// TwinCAT 3 PLC project PLC2
// ProgramVersion: 3.1.4024.0
// libraries:
//   Tc2_Standard, * (Beckhoff Automation GmbH)
//   Tc2_System, * (Beckhoff Automation GmbH)
//   Tc3_Module, * (Beckhoff Automation GmbH)
// project tree:
//   GVLs/ GVL_Alarm.TcGVL
//   / PlcTask.TcTTO
//   POUs/ Fb_AdsReader.TcPOU, FB_AlarmController.TcPOU, MAIN.TcPOU
// (motion and I/O tree: see PLC project plc1)
// real-time tasks:
//   TASK PlcTask: cycle T#10ms, priority 20, ADS port 350
//   TASK PlcTask1: cycle T#10ms, priority 21, ADS port 351

CONFIGURATION PLC2
    RESOURCE PLC ON TwinCAT3
        TASK PlcTask(INTERVAL := T#10ms, PRIORITY := 21);
        PROGRAM MAIN WITH PlcTask : MAIN;
    END_RESOURCE
END_CONFIGURATION

// ---- GVLs/GVL_Alarm.TcGVL
{attribute 'qualified_only'}
{attribute 'TcAdsSymEntry'}
VAR_GLOBAL
    // ── Values READ from PLC1 ────────────────────────────────────────
    nTankLevel      : INT;
    bOverflow       : BOOL;
    bUnderflow      : BOOL;
    sStatusMsg      : STRING;

    // ── Alarm panel variables (PLC2 own logic) ───────────────────────
    bAlarmActive    : BOOL;
    sAlarmMessage   : STRING := 'No Alarms';
    bAckAlarm       : BOOL;       // HMI operator presses this
END_VAR

// ---- POUs/MAIN.TcPOU
PROGRAM MAIN
VAR
	 fbAlarm : FB_AlarmController;
END_VAR

fbAlarm();

END_PROGRAM

// ---- POUs/FB_AlarmController.TcPOU
FUNCTION_BLOCK FB_AlarmController
VAR
    // ── ADS Readers — one per variable ──────────────────────────────
    fbReadLevel     : FB_AdsReader;
    fbReadOverflow  : FB_AdsReader;
    fbReadUnderflow : FB_AdsReader;
    fbReadStatus    : FB_AdsReader;
END_VAR


// ── Read nTankLevel from PLC1 every 500ms ────────────────────────────
fbReadLevel(
    sSymbol     := 'GVL_Tank.nTankLevel',
    nPort       := 851,
    tCycleTime  := T#500MS,
    pDestAddr   := ADR(GVL_Alarm.nTankLevel),
    nDestSize   := SIZEOF(GVL_Alarm.nTankLevel)
);

// ── Read bOverflow from PLC1 every 500ms ─────────────────────────────
fbReadOverflow(
    sSymbol     := 'GVL_Tank.bOverflow',
    nPort       := 851,
    tCycleTime  := T#500MS,
    pDestAddr   := ADR(GVL_Alarm.bOverflow),
    nDestSize   := SIZEOF(GVL_Alarm.bOverflow)
);

// ── Read bUnderflow from PLC1 every 500ms ────────────────────────────
fbReadUnderflow(
    sSymbol     := 'GVL_Tank.bUnderflow',
    nPort       := 851,
    tCycleTime  := T#500MS,
    pDestAddr   := ADR(GVL_Alarm.bUnderflow),
    nDestSize   := SIZEOF(GVL_Alarm.bUnderflow)
);

// ── Read sStatusMsg from PLC1 every 1s ───────────────────────────────
fbReadStatus(
    sSymbol     := 'GVL_Tank.sStatusMsg',
    nPort       := 851,
    tCycleTime  := T#1S,
    pDestAddr   := ADR(GVL_Alarm.sStatusMsg),
    nDestSize   := SIZEOF(GVL_Alarm.sStatusMsg)
);

// ── Alarm logic based on received values ─────────────────────────────
IF GVL_Alarm.bOverflow THEN
    GVL_Alarm.bAlarmActive  := TRUE;
    GVL_Alarm.sAlarmMessage := 'CRITICAL — Tank Overflow Detected';

ELSIF GVL_Alarm.bUnderflow THEN
    GVL_Alarm.bAlarmActive  := TRUE;
    GVL_Alarm.sAlarmMessage := 'WARNING — Tank Underflow Detected';

ELSE
    GVL_Alarm.bAlarmActive  := FALSE;
    GVL_Alarm.sAlarmMessage := 'No Alarms';
END_IF

END_FUNCTION_BLOCK

// ---- POUs/Fb_AdsReader.TcPOU
FUNCTION_BLOCK FB_AdsReader
VAR_INPUT
    sSymbol         : STRING;       // Symbol name to read e.g. 'GVL_Tank.nTankLevel'
    nPort           : UINT;         // Target PLC port e.g. 851
    tCycleTime      : TIME;         // How often to read e.g. T#500MS
    pDestAddr       : POINTER TO BYTE; // Pointer to local variable
    nDestSize       : UDINT;        // Size of local variable
END_VAR
VAR_OUTPUT
    bBusy           : BOOL;
    bError          : BOOL;
    nErrId          : UDINT;
    bNewValue       : BOOL;         // Pulses TRUE when fresh value arrives
END_VAR
VAR
    fbAdsRead       : ADSREAD;
    fbCycleTimer    : TON;
    bTrigger        : BOOL;
    bLastBusy       : BOOL;
END_VAR



// ── Cycle timer — fires every tCycleTime ─────────────────────────────
fbCycleTimer(IN := NOT fbCycleTimer.Q, PT := tCycleTime);

// ── Trigger a new read when timer fires and not already busy ─────────
IF fbCycleTimer.Q AND NOT bBusy THEN
    bTrigger := TRUE;
ELSE
    bTrigger := FALSE;
END_IF

// ── Execute ADSREAD ──────────────────────────────────────────────────
fbAdsRead(
    NETID    := '',
    PORT     := nPort,
    IDXGRP   := 16#F005,
    IDXOFFS  := TO_UDINT(ADR(sSymbol)),
    LEN      := nDestSize,
    DESTADDR := pDestAddr,
    READ     := bTrigger,
    BUSY     => bBusy,
    ERR      => bError,
    ERRID    => nErrId
);

// ── bNewValue pulses TRUE for one scan when read completes ───────────
bNewValue := bLastBusy AND NOT bBusy AND NOT bError;
bLastBusy := bBusy;

END_FUNCTION_BLOCK
